// TIA Portal project "MiscelatoreFB" (V16)

(* hardware
DEVICE "S7-1200 station_1"  S7-1200 Station
   slot 0: "Telaio di montaggio_0"  S7-1200 Rack  Rack  V1.0
   slot 1: "PLC_1"  CPU 1214C DC/DC/DC  6ES7 214-1AG40-0XB0  V4.1
*)

// ===== PLC "PLC_1"  CPU 1214C DC/DC/DC =====

VAR_GLOBAL   // PLC tag table "Tabella delle variabili standard"
   "START" AT %I0.0 : Bool;
   "FULL_SENSOR" AT %I0.1 : Bool;
   "EMPTY_SENSOR" AT %I0.2 : Bool;
   "SOL_A" AT %Q0.0 : Bool;
   "SOL_B" AT %Q0.1 : Bool;
   "MOTOR" AT %Q0.2 : Bool;
   "RESISTOR" AT %Q0.3 : Bool;
END_VAR

VAR_GLOBAL CONSTANT   // PLC tag table "Tabella delle variabili standard"
   "TEMPO_TRASCORSO_T1" : Time := T#30s;
   "TEMPO_TRASCORSO_T2" : Time := T#15s;
END_VAR

DATA_BLOCK "Misceltatore_DB"   // DB1
{ S7_Optimized_Access := 'TRUE' }
VERSION : 0.1
// stored: InstanceOfName Misceltatore
"Misceltatore"
BEGIN
END_DATA_BLOCK

FUNCTION_BLOCK "Misceltatore"   // FB1, LAD
{ S7_Optimized_Access := 'TRUE' }
VERSION : 0.1
   VAR_INPUT
      START : Bool;
      FULL_SENSOR : Bool;
      EMPTY_SENSOR : Bool;
      TEMPO_TRASCORSO_T1 : Time;
      TEMPO_TRASCORSO_T2 : Time;
   END_VAR
   VAR_OUTPUT
      SOL_A : Bool;
      SOL_B : Bool;
      MOTOR : Bool;
      RESISTOR : Bool;
   END_VAR
   VAR RETAIN
      HOME : Bool := true;
   END_VAR
   VAR
      OPEN_SOL_A : Bool;
   END_VAR
   VAR RETAIN
      CLOSE_SOL_A : Bool;
      INACTIVITY_STATE : Bool;
      ACTIVITY_STATE : Bool;
      OPEN_SOL_B : Bool;
   END_VAR
   VAR
      IEC_Timer_0_Instance_1 : TON_TIME;
      IEC_Timer_0_Instance_2 : TON_TIME;
      IEC_Timer_0_Instance_3 : TON_TIME;
   END_VAR
BEGIN

REGION Network 1
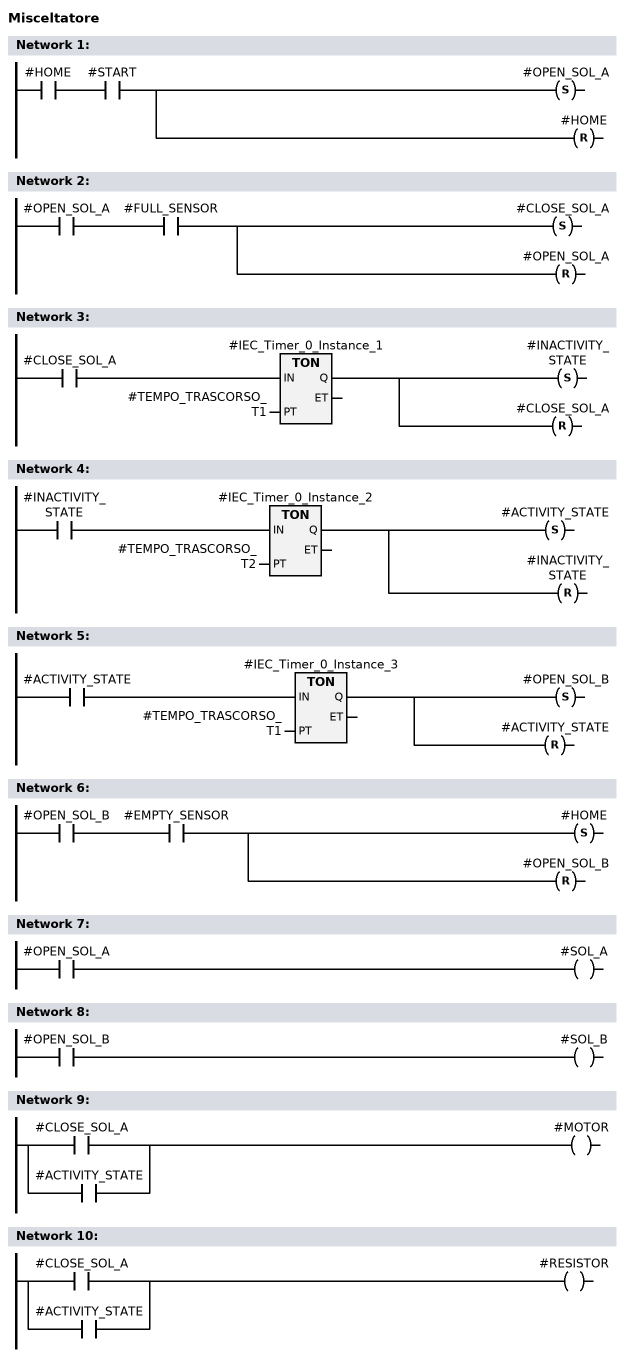
   RUNG wire#powerrail
      Contact( #HOME )
      Contact( #START )
      wire#w1
      S_Coil( #OPEN_SOL_A )
   END_RUNG
   RUNG wire#w1
      R_Coil( #HOME )
   END_RUNG
   // the same network as SCL:
   IF #HOME AND #START THEN
       #OPEN_SOL_A := TRUE;
       #HOME := FALSE;
   END_IF;
END_REGION

REGION Network 2
   RUNG wire#powerrail
      Contact( #OPEN_SOL_A )
      Contact( #FULL_SENSOR )
      wire#w1
      S_Coil( #CLOSE_SOL_A )
   END_RUNG
   RUNG wire#w1
      R_Coil( #OPEN_SOL_A )
   END_RUNG
   // the same network as SCL:
   IF #OPEN_SOL_A AND #FULL_SENSOR THEN
       #CLOSE_SOL_A := TRUE;
       #OPEN_SOL_A := FALSE;
   END_IF;
END_REGION

REGION Network 3
   #IEC_Timer_0_Instance_1(IN := #CLOSE_SOL_A, PT := #TEMPO_TRASCORSO_T1);   // TON
   IF #IEC_Timer_0_Instance_1.Q THEN
       #INACTIVITY_STATE := TRUE;
       #CLOSE_SOL_A := FALSE;
   END_IF;
END_REGION

REGION Network 4
   #IEC_Timer_0_Instance_2(IN := #INACTIVITY_STATE, PT := #TEMPO_TRASCORSO_T2);   // TON
   IF #IEC_Timer_0_Instance_2.Q THEN
       #ACTIVITY_STATE := TRUE;
       #INACTIVITY_STATE := FALSE;
   END_IF;
END_REGION

REGION Network 5
   #IEC_Timer_0_Instance_3(IN := #ACTIVITY_STATE, PT := #TEMPO_TRASCORSO_T1);   // TON
   IF #IEC_Timer_0_Instance_3.Q THEN
       #OPEN_SOL_B := TRUE;
       #ACTIVITY_STATE := FALSE;
   END_IF;
END_REGION

REGION Network 6
   RUNG wire#powerrail
      Contact( #OPEN_SOL_B )
      Contact( #EMPTY_SENSOR )
      wire#w1
      S_Coil( #HOME )
   END_RUNG
   RUNG wire#w1
      R_Coil( #OPEN_SOL_B )
   END_RUNG
   // the same network as SCL:
   IF #OPEN_SOL_B AND #EMPTY_SENSOR THEN
       #HOME := TRUE;
       #OPEN_SOL_B := FALSE;
   END_IF;
END_REGION

REGION Network 7
   RUNG wire#powerrail
      Contact( #OPEN_SOL_A )
      Coil( #SOL_A )
   END_RUNG
   // the same network as SCL:
   #SOL_A := #OPEN_SOL_A;
END_REGION

REGION Network 8
   RUNG wire#powerrail
      Contact( #OPEN_SOL_B )
      Coil( #SOL_B )
   END_RUNG
   // the same network as SCL:
   #SOL_B := #OPEN_SOL_B;
END_REGION

REGION Network 9
   RUNG wire#powerrail
      Contact( #CLOSE_SOL_A )
      wire#w1
      Coil( #MOTOR )
   END_RUNG
   RUNG wire#powerrail
      Contact( #ACTIVITY_STATE )
   END_RUNG wire#w1
   // the same network as SCL:
   #MOTOR := #CLOSE_SOL_A OR #ACTIVITY_STATE;
END_REGION

REGION Network 10
   RUNG wire#powerrail
      Contact( #CLOSE_SOL_A )
      wire#w1
      Coil( #RESISTOR )
   END_RUNG
   RUNG wire#powerrail
      Contact( #ACTIVITY_STATE )
   END_RUNG wire#w1
   // the same network as SCL:
   #RESISTOR := #CLOSE_SOL_A OR #ACTIVITY_STATE;
END_REGION
END_FUNCTION_BLOCK

ORGANIZATION_BLOCK "Main"   // OB1, LAD, ProgramCycle
TITLE = "Main Program Sweep (Cycle)"
{ S7_Optimized_Access := 'TRUE' }
VERSION : 0.1
   VAR_INPUT
      Initial_Call : Bool;   // Initial call of this OB
      Remanence : Bool;   // =True, if remanent data are available
   END_VAR
BEGIN
END_ORGANIZATION_BLOCK

ORGANIZATION_BLOCK "Cyclic_Interrupt_50ms"   // OB30, LAD, CyclicInterrupt
{ S7_Optimized_Access := 'TRUE' }
VERSION : 0.1
   VAR_INPUT
      Initial_Call : Bool;   // Initial call of this OB
      Event_Count : Int;   // Events discarded
   END_VAR
BEGIN

REGION Network 1
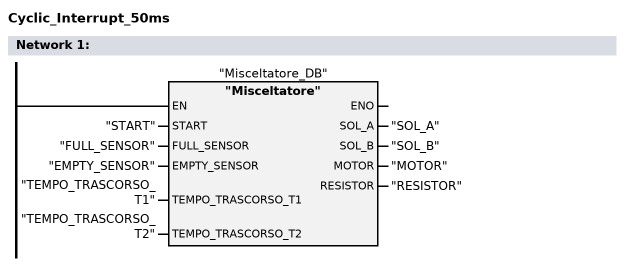
   RUNG wire#powerrail
      "Misceltatore_DB"(START := "START", FULL_SENSOR := "FULL_SENSOR", EMPTY_SENSOR := "EMPTY_SENSOR", TEMPO_TRASCORSO_T1 := "TEMPO_TRASCORSO_T1", TEMPO_TRASCORSO_T2 := "TEMPO_TRASCORSO_T2", SOL_A => "SOL_A", SOL_B => "SOL_B", MOTOR => "MOTOR", RESISTOR => "RESISTOR")
   END_RUNG
   // the same network as SCL:
   "Misceltatore_DB"(START := "START",   // "Misceltatore"
                     FULL_SENSOR := "FULL_SENSOR",
                     EMPTY_SENSOR := "EMPTY_SENSOR",
                     TEMPO_TRASCORSO_T1 := "TEMPO_TRASCORSO_T1",
                     TEMPO_TRASCORSO_T2 := "TEMPO_TRASCORSO_T2",
                     SOL_A => "SOL_A",
                     SOL_B => "SOL_B",
                     MOTOR => "MOTOR",
                     RESISTOR => "RESISTOR");
END_REGION
END_ORGANIZATION_BLOCK